(* IEC 61131-3 sources: SmartHouseIOT/, 8 files *)

(* ---- 06_IOT_HOUSE.ST ---- *)
VAR_GLOBAL
  //system
  timePLC AT %s16 : INT;
  timeDelayed : INT := 0;
  switchCase : INT := 0;
  // lights
  bedroomLight : BOOL := FALSE;
  childTopRoomLight : BOOL := FALSE;
  garageLight : BOOL := FALSE;
  childMiddleRoomLight : BOOL := FALSE;
  bathroomLight : BOOL := FALSE;
  hallLight : BOOL := FALSE;
  wcLight : BOOL := FALSE;
  kitchenLight : BOOL := FALSE;
  patioLight : BOOL := FALSE;
  livingRoomLight : BOOL := FALSE;
  outsideLight : BOOL := FALSE;
  cellarLight : BOOL := FALSE;
  //sun
  sun : BOOL := FALSE;
  cycleSwitched : BOOL := FALSE;
  // doors
  bedroomDoor : BOOL := FALSE;
  childTopRoomDoor : BOOL := FALSE;
  childMiddleRoomDoor : BOOL := FALSE;
  garageDoor : BOOL := FALSE;
  garageGate : BOOL := FALSE;
  bathroomDoor : BOOL := FALSE;
  wcDoor : BOOL := FALSE;
  cellarDoor : BOOL := FALSE;
  patioDoor : BOOL := FALSE;
  hallDoor : BOOL := FALSE;
  // info text
  insideTemperatureText : STRING := '';
  outsideTemperatureText : STRING := '';
  // master password
  MASTER_PASSKEY : STRING := '1234';
  // security
  enteredPassKey : STRING := '';
  enteredPassKeyINT : INT := 0;
  enteredPassKeyINTdefaultValue : INT := 0;
  canOpenOutsideDoors : BOOL := FALSE;
  alarmON : BOOL := FALSE;
  alarmBlink : BOOl := FALSE;
  passKeyDefaultValue : STRING := '';
  alarmTimerOFFsec : INT := 0;
  defaultAlarmTimerOFFsec : INT := 5;
  // temperature
  insideTemperature : DINT := 10;
  heating : BOOL := FALSE;
  outsideTemperature : DINT := 15;
  DESIRED_TEMPERATURE : DINT := 21;
  cooling : BOOL := FALSE;
  // master switches
  masterLightSwitchON : BOOL := FALSE;
  masterLightSwitchOFF : BOOL := FALSE;
  // switches
  bedroomLightSwitch : BOOL := FALSE;
  childTopRoomLightSwitch : BOOL := FALSE;
  garageLightSwitch : BOOL := FALSE;
  childMiddleRoomLightSwitch : BOOL := FALSE;
  bathroomLightSwitch : BOOL := FALSE;
  hallLightSwitch : BOOL := FALSE;
  wcLightSwitch : BOOL := FALSE;
  kitchenLightSwitch : BOOL := FALSE;
  patioLightSwitch : BOOL := FALSE;
  livingRoomLightSwitch : BOOL := FALSE;
  outsideLightSwitch : BOOL := FALSE;
  cellarLightSwitch : BOOL := FALSE;
  garageGateSwitch : BOOL := FALSE;
  garageDoorSwitch : BOOL := FALSE;
  frontDoorSwitch : BOOL := FALSE;
  patioDoorSwitch : BOOL := FALSE;
  // misc
  secsInMin : INT := 6;
  modTime : INT := 0;
  modTemp : DINT := 0;
  random : BOOL := FALSE;
  canCallTemperatureChange : BOOL := FALSE;
  textAllON : STRING := 'All ON';
  textAllOFF : STRING := 'All OFF';
  textOutsideLights : STRING := 'Outside lights';
  textPassKey : STRING := 'PassKey:';
  textLights : STRING := 'Lights Controller';
  textSecuritySystem : STRING := 'Security Controller';
  // PRNG
  seed: DINT := 123;  // Initial seed value
  a: DINT := 1664525; // Multiplier
  c: DINT := 1013904223; // Increment
  m: DINT := 2147483647; // Modulus (2^31)
  randomValue: DINT;
END_VAR

(* ---- HandleDayNightCycle.ST ---- *)
FUNCTION HandleDayNightCycle : BOOL
  VAR_INPUT
  END_VAR
  VAR_IN_OUT
  END_VAR
  VAR
  END_VAR
  VAR_TEMP
  END_VAR

  modTime := timePLC MOD secsInMin;
  IF modTime = 0 AND NOT cycleSwitched THEN
    cycleSwitched := TRUE;
    IF sun THEN
      sun := FALSE;
    ELSE
      sun := TRUE;
    END_IF;
    canCallTemperatureChange := TRUE;
  ELSIF modTime = 0 AND cycleSwitched THEN
    canCallTemperatureChange := FALSE;
  ELSE
    cycleSwitched := false;
    canCallTemperatureChange := FALSE;
  END_IF;
END_FUNCTION

(* ---- HandleLights.ST ---- *)
FUNCTION HandleLights : BOOL
  VAR_INPUT
  END_VAR
  VAR_IN_OUT
  END_VAR
  VAR
  END_VAR
  VAR_TEMP
  END_VAR

  IF masterLightSwitchOFF THEN
    bedroomLight         := FALSE;
    childTopRoomLight    := FALSE;
    garageLight          := FALSE;
    childMiddleRoomLight := FALSE;
    bathroomLight        := FALSE;
    hallLight            := FALSE;
    wcLight              := FALSE;
    kitchenLight         := FALSE;
    patioLight           := FALSE;
    livingRoomLight      := FALSE;
    outsideLight         := FALSE;
    cellarLight          := FALSE;
  ELSIF masterLightSwitchON THEN
    bedroomLight         := TRUE;
    childTopRoomLight    := TRUE;
    garageLight          := TRUE;
    childMiddleRoomLight := TRUE;
    bathroomLight        := TRUE;
    hallLight            := TRUE;
    wcLight              := TRUE;
    kitchenLight         := TRUE;
    patioLight           := TRUE;
    livingRoomLight      := TRUE;
    outsideLight         := TRUE;
    cellarLight          := TRUE;
  ELSE
    bedroomLight         := bedroomLightSwitch;
    childTopRoomLight    := childTopRoomLightSwitch;
    garageLight          := garageLightSwitch;
    childMiddleRoomLight := childMiddleRoomLightSwitch;
    bathroomLight        := bathroomLightSwitch;
    hallLight            := hallLightSwitch;
    wcLight              := wcLightSwitch;
    kitchenLight         := kitchenLightSwitch;
    patioLight           := patioLightSwitch;
    livingRoomLight      := livingRoomLightSwitch;
    cellarLight          := cellarLightSwitch;
    IF NOT SUN THEN
      outsideLight       := TRUE;
    ELSE
      outsideLight       := outsideLightSwitch;
    END_IF;
  END_IF;

END_FUNCTION

(* ---- HandleSecurity.ST ---- *)
FUNCTION HandleSecurity : BOOL
  VAR_INPUT
  END_VAR
  VAR_IN_OUT
  END_VAR
  VAR
  END_VAR
  VAR_TEMP
  END_VAR

  IF NOT enteredPassKey = passKeyDefaultValue THEN
    IF enteredPassKey = MASTER_PASSKEY THEN
      canOpenOutsideDoors := TRUE;
      alarmON := FALSE;
      alarmTimerOFFsec := defaultAlarmTimerOFFsec;
    ELSE
      alarmON := TRUE;
      canOpenOutsideDoors := FALSE;
    END_IF;
    enteredPassKey := passKeyDefaultValue;
  END_IF;

  IF NOT enteredPassKeyINT = enteredPassKeyINTdefaultValue THEN
    IF INT_TO_STRING(enteredPassKeyINT) = MASTER_PASSKEY THEN
      canOpenOutsideDoors := TRUE;
      alarmON := FALSE;
      alarmTimerOFFsec := defaultAlarmTimerOFFsec;
    ELSE
      alarmON := TRUE;
      canOpenOutsideDoors := FALSE;
    END_IF;
    enteredPassKey := passKeyDefaultValue;
    enteredPassKeyINT := 0;
  END_IF;

  IF canOpenOutsideDoors THEN
    garageGate := garageGateSwitch;
    garageDoor := garageDoorSwitch;
    patioDoor  := patioDoorSwitch;
    hallDoor   := frontDoorSwitch;
  ELSE
    garageGate := FALSE;
    garageDoor := FALSE;
    patioDoor  := FALSE;
    hallDoor   := FALSE;

    garageGateSwitch := FALSE;
    garageDoorSwitch := FALSE;
    patioDoorSwitch  := FALSE;
    frontDoorSwitch  := FALSE;
  END_IF;

END_FUNCTION

(* ---- HandleTemperature.ST ---- *)
FUNCTION HandleTemperature : BOOL
  VAR_INPUT
  END_VAR
  VAR_IN_OUT
  END_VAR
  VAR
  seedAbs : DINT := 0;
  END_VAR
  VAR_TEMP
  END_VAR

  seedAbs := ABS(seed);
  IF sun THEN
    outsideTemperature := outsideTemperature + (seedAbs MOD 3);
  ELSE
    outsideTemperature := outsideTemperature - (seedAbs MOD 3);
  END_IF;
  insideTemperature := (insideTemperature + outsideTemperature) / 2;//insideTemperature + ((insideTemperature - outsideTemperature) / 2);

  IF insideTemperature = DESIRED_TEMPERATURE THEN
    heating := FALSE;
    cooling := FALSE;
  ELSIF insideTemperature < DESIRED_TEMPERATURE THEN
    heating := TRUE;
    cooling := FALSE;
    insideTemperature := insideTemperature + 3;
  ELSE
    cooling := TRUE;
    heating := FALSE;
    insideTemperature := insideTemperature - 3;
  END_IF;

END_FUNCTION

(* ---- PRNG.ST ---- *)
FUNCTION PRNG : DINT
  VAR_INPUT
  END_VAR
  VAR_IN_OUT
  END_VAR
  VAR
  END_VAR
  VAR_TEMP
  END_VAR

  seed := a * seed;
  seed := seed + c;
  seed := seed MOD m;
  RETURN;
END_FUNCTION

(* ---- Test.ST ---- *)
FUNCTION Test : BOOL
  VAR_INPUT
  END_VAR
  VAR_IN_OUT
  END_VAR
  VAR
  END_VAR
  VAR_TEMP
  END_VAR
END_FUNCTION

(* ---- prgMain.ST ---- *)
PROGRAM prgMain
  VAR_INPUT
  END_VAR
  VAR_OUTPUT
  END_VAR
  VAR
  END_VAR
  VAR_TEMP
  END_VAR

  PRNG();
  modTemp := seed;
  modTemp := modTemp MOD 2;
  PRNG();
  random := seed < 0;
  HandleLights();

  HandleDayNightCycle();
  IF canCallTemperatureChange THEN
  END_IF;
  insideTemperatureText := DINT_TO_STRING(insideTemperature) + ' °C';
  outsideTemperatureText := DINT_TO_STRING(outsideTemperature) + ' °C';

  CASE switchCase OF
    0:
      IF timePLC >= timeDelayed THEN
        HandleTemperature();
        switchCase := 1;

        IF alarmTimerOFFsec > 0 THEN
          alarmTimerOFFsec := alarmTimerOFFsec - 1;
        ELSE
          canOpenOutsideDoors := FALSE;
        END_IF;

      END_IF;
    1:
      timeDelayed := timePLC + 1;
      switchCase := 0;

      IF alarmON THEN
        IF alarmBlink THEN
          alarmBlink := FALSE;
        ELSE
          alarmBlink := TRUE;
        END_IF;
      ELSE
        alarmBlink := FALSE;
      END_IF;
  END_CASE;

  HandleSecurity();
END_PROGRAM
